FUNCTION_BLOCK MockInit IMPLEMENTS I_Initialisable, I_Object
VAR
	_isRegistered : BOOL;
END_VAR

METHOD Initialise : HRESULT
END_METHOD

{warning 'Add property implementation'}
PROPERTY Initialised : BOOL
GET
Initialised := TRUE;
END_GET
END_PROPERTY

METHOD IsRegistered : BOOL
VAR_INPUT
END_VAR
IsRegistered := _isRegistered;
END_METHOD

METHOD RegisterWithParent
VAR_INPUT
	Parent	: I_HostObjects;
END_VAR
IF NOT _isRegistered THEN
	IF SUCCEEDED(Parent.RegisterInitialisable(THIS^)) THEN
		_isRegistered := TRUE;
	ELSE
		_isRegistered := FALSE;
	END_IF
END_IF
END_METHOD

END_FUNCTION_BLOCK

(* stored: Version 1.1.0.1
   POU MockInit: Id {ea0d0635-4bc8-4e40-bb70-64fdc548ef76}, SpecialFunc None
   Method Initialise: Id {93202d8c-ca65-49f4-bc1a-ba79c2f00c97}
   Property Initialised: Id {8eca6b5f-e7d9-48fd-a262-c4eb08cb3a85}
   Get Get: Id {b0a04522-1f9a-44e9-8852-891b0f1a43ae}
   Method IsRegistered: Id {0cc4c4a8-8a78-4ee1-b5e7-9370aa13080b}
   Method RegisterWithParent: Id {8a07062e-82db-456a-9ee2-ded9fd286a71} *)
